// TIA Portal project "progetto1" (V16)

(* hardware
DEVICE "S7-1200 station_1"  S7-1200 Station
   slot 0: "Rack_0"  S7-1200 Rack  Rack  V1.0
   slot 1: "PLC_1"  CPU 1212C DC/DC/DC  6ES7 212-1AE40-0XB0  V4.4
   slot 2: "DI 8/DQ 8x24VDC_1"  6ES7 223-1BH32-0XB0  V2.0
*)

// ===== PLC "PLC_1"  CPU 1212C DC/DC/DC =====

VAR_GLOBAL   // PLC tag table "Default tag table"
   "PULSANTE EMERGENZA" AT %M2.0 : Bool;
   "INPUT START" AT %I1.3 : Bool;
   "INPUT STOP" AT %I1.4 : Bool;
   "INPUT EMERGENZA" AT %I1.0 : Bool;
   "INPUT SELETTORE MAN/AUTO" AT %I1.5 : Bool;
   "INPUT RESET EMERGENZA" AT %I1.1 : Bool;
   "INPUT PULSANTE 1" AT %I1.2 : Bool;
   "INPUT PULSANTE 3" AT %I1.7 : Bool;
   "INPUT PULSANTE 2" AT %I1.6 : Bool;
   "O PINZA ROBOT EV" AT %Q1.7 : Bool;
   "O ROBOT SINISTRA/DESTRA EV" AT %Q1.6 : Bool;
   "O ROBOT SU E GIU EV" AT %Q1.5 : Bool;
   "O ROBOT AVANTI E INDIETRO EV" AT %Q1.4 : Bool;
   "O LAMPADA START" AT %Q1.3 : Bool;
   "O SPIA/LAMPADA RESET EMERGENZA" AT %Q1.2 : Bool;
   "SENSORE ROBOT DESTRA" AT %I0.5 : Bool;
   "SENSORE ROBOT SINISTRA" AT %I0.4 : Bool;
   "SENSORE ROBOT GIU" AT %I0.2 : Bool;
   "SENSORE ROBOT SU" AT %I0.3 : Bool;
   "SENSORE ROBOT AVANTI" AT %I0.0 : Bool;
   "SENSORE ROBOT INDIETRO" AT %I0.1 : Bool;
   "System_Byte" AT %MB1 : Byte;
   "FirstScan" AT %M1.0 : Bool;
   "DiagStatusUpdate" AT %M1.1 : Bool;
   "AlwaysTRUE" AT %M1.2 : Bool;
   "AlwaysFALSE" AT %M1.3 : Bool;
   "Clock_Byte" AT %MB0 : Byte;
   "Clock_10Hz" AT %M0.0 : Bool;
   "Clock_5Hz" AT %M0.1 : Bool;
   "Clock_2.5Hz" AT %M0.2 : Bool;
   "Clock_2Hz" AT %M0.3 : Bool;
   "Clock_1.25Hz" AT %M0.4 : Bool;
   "Clock_1Hz" AT %M0.5 : Bool;
   "Clock_0.625Hz" AT %M0.6 : Bool;
   "Clock_0.5Hz" AT %M0.7 : Bool;
END_VAR

DATA_BLOCK "HMI_IMPIANTO"   // DB1
{ S7_Optimized_Access := 'TRUE' }
VERSION : 0.1
   VAR
      OUT_LOCAL_STATE : Int;
   END_VAR
BEGIN
END_DATA_BLOCK

DATA_BLOCK "STATI_IMPIANTO"   // DB2
{ S7_Optimized_Access := 'TRUE' }
VERSION : 0.1
   VAR
      "COMANDO ROBOT SINISTRA" : Bool;
      "COMANDO ROBOT SU" : Bool;
      "COMANDO ROBOT AVANTI7" : Bool;
      "COMANDO ROBOT PINZA CHIUSA" : Bool;
   END_VAR
BEGIN
END_DATA_BLOCK

FUNCTION "COMANDI ROBOT" : Void   // FC1, SCL
{ S7_Optimized_Access := 'TRUE' }
VERSION : 0.1
BEGIN

   IF "INPUT PULSANTE 1" THEN

       "O ROBOT AVANTI E INDIETRO EV" := "Clock_10Hz";
   END_IF;
END_FUNCTION

FUNCTION "APRI CHIUDI ROBOT" : Void   // FC2, SCL
{ S7_Optimized_Access := 'TRUE' }
VERSION : 0.1
BEGIN
   IF  "INPUT RESET EMERGENZA" THEN
       "O ROBOT SU E GIU EV" := 0;
       "O ROBOT SINISTRA/DESTRA EV" := 0;
       "O ROBOT SU E GIU EV" := 0;
       "O PINZA ROBOT EV" := 0;
   ELSE
       IF "INPUT PULSANTE 1" THEN
       // Statement section IF


       IF "SENSORE ROBOT AVANTI" THEN
           "O ROBOT AVANTI E INDIETRO EV" := 0;
           ;
       END_IF;
       IF "SENSORE ROBOT INDIETRO" THEN
           "O ROBOT AVANTI E INDIETRO EV" := 1;
          ;
      END_IF;

       IF "SENSORE ROBOT DESTRA" THEN
           "O ROBOT SINISTRA/DESTRA EV" := 1;
           ;
       END_IF;
       IF "SENSORE ROBOT SINISTRA" THEN
           "O ROBOT SINISTRA/DESTRA EV" := 0;
           ;
       END_IF;

       IF "SENSORE ROBOT GIU" THEN
           "O ROBOT SU E GIU EV" := 1;
           "O PINZA ROBOT EV" := 1;
           ;
       END_IF;
       IF "SENSORE ROBOT SU" THEN
           "O ROBOT SU E GIU EV" := 0;
           "O PINZA ROBOT EV" := 0;
           ;
       END_IF;
       ;
   END_IF;

   END_IF;
END_FUNCTION

FUNCTION "AUTOMATICO" : Void   // FC3, SCL
{ S7_Optimized_Access := 'TRUE' }
VERSION : 0.1
BEGIN

   IF NOT "INPUT SELETTORE MAN/AUTO" OR NOT "INPUT EMERGENZA" THEN
       "STATI_IMPIANTO"."COMANDO ROBOT AVANTI7" := FALSE;
       "STATI_IMPIANTO"."COMANDO ROBOT PINZA CHIUSA" := FALSE;
       "STATI_IMPIANTO"."COMANDO ROBOT SINISTRA" := FALSE;
       "STATI_IMPIANTO"."COMANDO ROBOT SU" := FALSE;
       "HMI_IMPIANTO".OUT_LOCAL_STATE := 0;
   END_IF;


   CASE "HMI_IMPIANTO".OUT_LOCAL_STATE OF


      0:  // Inizio sequenza (Vado su)
          IF "INPUT SELETTORE MAN/AUTO"
              AND "SENSORE ROBOT DESTRA"
              AND "SENSORE ROBOT GIU"
              AND "SENSORE ROBOT INDIETRO"
              AND "INPUT START"
          THEN
              "STATI_IMPIANTO"."COMANDO ROBOT SU" := TRUE;
              "HMI_IMPIANTO".OUT_LOCAL_STATE := 1;
          END_IF;
      1:  // Controllo su feedback e vado a sinistra
          IF "SENSORE ROBOT DESTRA"
              AND "SENSORE ROBOT SU"
              AND "SENSORE ROBOT INDIETRO"
          THEN
              "STATI_IMPIANTO"."COMANDO ROBOT SINISTRA":=TRUE;
              "HMI_IMPIANTO".OUT_LOCAL_STATE := 2;
          END_IF;
      2:  // Controllo sinistra feedback e vado avanti
          IF "SENSORE ROBOT SINISTRA"
              AND "SENSORE ROBOT SU"
              AND "SENSORE ROBOT INDIETRO"
          THEN
              "STATI_IMPIANTO"."COMANDO ROBOT AVANTI7" := TRUE;
              "HMI_IMPIANTO".OUT_LOCAL_STATE := 3;
          END_IF;
          3:  // Controllo feedback e chiudo pinza
              IF "SENSORE ROBOT SINISTRA"
                  AND "SENSORE ROBOT SU"
                  AND "SENSORE ROBOT AVANTI"
              THEN
                  "STATI_IMPIANTO"."COMANDO ROBOT PINZA CHIUSA" := TRUE;
              "HMI_IMPIANTO".OUT_LOCAL_STATE := 4;
          END_IF;
      4: //Controllo tutti i feedback
          IF "SENSORE ROBOT SINISTRA"
              AND "SENSORE ROBOT SU"
              AND "SENSORE ROBOT AVANTI"
          THEN
              "HMI_IMPIANTO".OUT_LOCAL_STATE :=5 ;
          END_IF;

          5: //fine sequenza
              ;
   END_CASE;
END_FUNCTION

FUNCTION "COMANDO_OUTPUT" : Void   // FC4, LAD
{ S7_Optimized_Access := 'TRUE' }
VERSION : 0.1
BEGIN

REGION Network 2 (SCL)
   "O PINZA ROBOT EV" := "STATI_IMPIANTO"."COMANDO ROBOT PINZA CHIUSA";
   "O ROBOT AVANTI E INDIETRO EV" := "STATI_IMPIANTO"."COMANDO ROBOT AVANTI7";
   "O ROBOT SU E GIU EV" := "STATI_IMPIANTO"."COMANDO ROBOT SU";
   "O ROBOT SINISTRA/DESTRA EV" := "STATI_IMPIANTO"."COMANDO ROBOT SINISTRA";
END_REGION
END_FUNCTION

ORGANIZATION_BLOCK "Main"   // OB1, LAD, ProgramCycle
TITLE = "Main Program Sweep (Cycle)"
{ S7_Optimized_Access := 'TRUE' }
VERSION : 0.1
   VAR_INPUT
      Initial_Call : Bool;   // Initial call of this OB
      Remanence : Bool;   // =True, if remanent data are available
   END_VAR
BEGIN

REGION Network 2 (SCL)
   "AUTOMATICO"();
   "COMANDO_OUTPUT"();
END_REGION
END_ORGANIZATION_BLOCK